{attribute 'qualified_only'}
{attribute 'strict'}
TYPE
ST100_Load_e :
(
    RESET := 0,         // Reset
    INIT := 100,        // Initialisieren 
    READY := 999,       // READY to Start, Init Done 
    START := 1000,      // Start Zyklisch
    MOVER_FREE_OP,      // Ab here, operation without mover can be done
    proceedOperation_1, // proceed to some operation
    waitOnMover,        // wait until the mover is there
    MOVER_NEEDED_OP,    // Ab here, a mover in position is needed to perform the action
    proceedOperation_2, // proceed to some operation
    SYNC_MOVER_LEAVE,   // MoverMan need to take the mover
    DONE := 8000,       // Ablauf beendet 
    ERROR := 9000,      // Fehler 
    _max
);
END_TYPE

(* stored: Version 1.1.0.1, ProductVersion 3.1.4024.6
   EnumerationTextList ST100_Load_e: Id {ab163a4a-f24e-4f30-889f-e72618526d74} *)
